TYPE PuckLnSw :
STRUCT
	///DB Input
	RFID: DINT;
	///DB Input
	Location: STRING(30);
	///DB Output
	PrimaryLane: STRING(30);
	///DB Output
	SecondaryLane: STRING(30);
	///DB Output
	TertiaryLane: STRING(30);
	///DB Output
	PuckSide: STRING(30);
	///DB Output
	IsHighPriority: BOOL;
	///PLC Internal variable
	InfeedBelt: DINT;
	///PLC Internal variable
	OutfeedDivert: DINT;
	///PLC Internal variable
	TransferStage: DINT;
END_STRUCT
END_TYPE

(* stored: Version 1.1.0.1, ProductVersion 3.1.4024.6
   DUT PuckLnSw: Id {4857292d-fcc6-4b78-be77-3f6a1fbf00b2} *)
